// Mitsubishi GX Works2 project: 시퀀스 연속동작, 단속동작   PLC: Q03UDV

PROGRAM MAIN
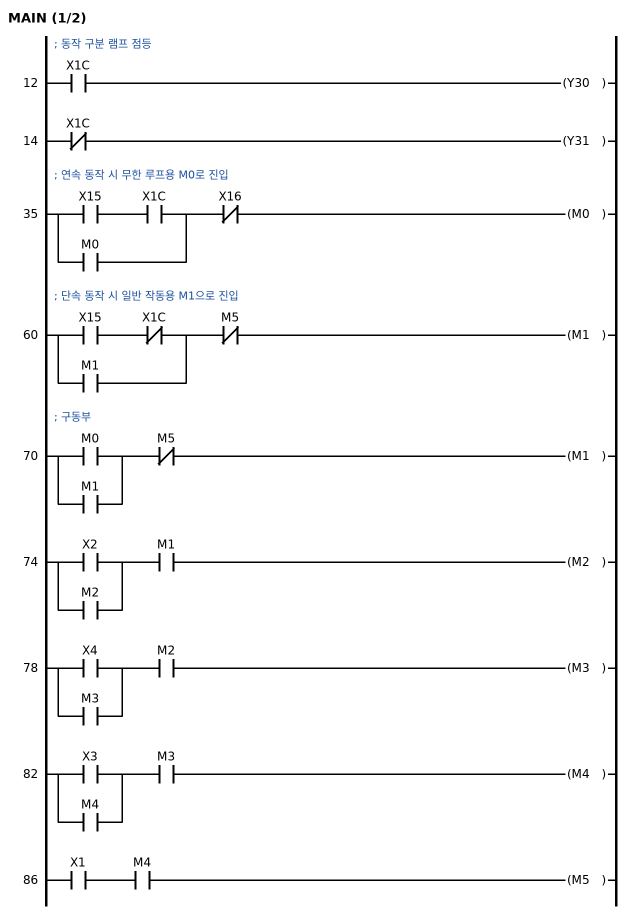
; 동작 구분 램프 점등
12    LD      X1C
      OUT     Y30
14    LDI     X1C
      OUT     Y31
; 연속 동작 시 무한 루프용 M0로 진입
35    LD      X15
      AND     X1C
      OR      M0
      ANI     X16
      OUT     M0
; 단속 동작 시 일반 작동용 M1으로 진입
60    LD      X15
      ANI     X1C
      OR      M1
      ANI     M5
      OUT     M1
; 구동부
70    LD      M0
      OR      M1
      ANI     M5
      OUT     M1
74    LD      X2
      OR      M2
      AND     M1
      OUT     M2
78    LD      X4
      OR      M3
      AND     M2
      OUT     M3
82    LD      X3
      OR      M4
      AND     M3
      OUT     M4
86    LD      X1
      AND     M4
      OUT     M5
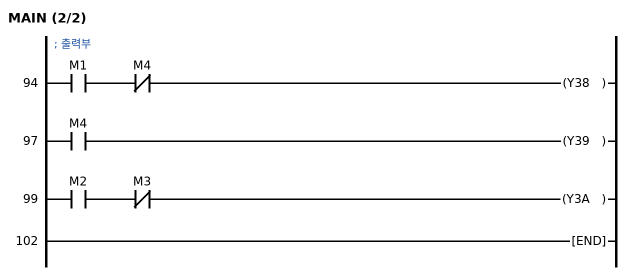
; 출력부
94    LD      M1
      ANI     M4
      OUT     Y38
97    LD      M4
      OUT     Y39
99    LD      M2
      ANI     M3
      OUT     Y3A
102   END
END_PROGRAM
